INTERFACE I_TraceInstanceLogger EXTENDS I_Base

METHOD LogMessageInstance
VAR_INPUT
	SourceInfo	: I_TraceSourceInfo;
	MessageInfo : I_TraceMessageInfo;
	Arguments	: I_TraceArgument := 0;
END_VAR
END_METHOD

END_INTERFACE

(* stored: Version 1.1.0.1, ProductVersion 3.1.4026.18
   Itf I_TraceInstanceLogger: Id {56419aad-3f86-0d19-244d-3b3b97f76f31}
   Method LogMessageInstance: Id {24b8b30c-f4be-0c4d-19e9-3553dacb32c1} *)
